(* IEC 61131-3 sources: verifaps-lib/share/PPU.stold (part 8) *)

(* ---- Scenario13_Final.xml_Pusher.st ---- *)
FUNCTION_BLOCK Pusher
    VAR  Duration2 : TIME := TIME#2.0s; END_VAR {*Lrwxp*}
    VAR  Duration3 : TIME := TIME#200.0ms; END_VAR {*Lrwxp*}
    VAR  Duration_Slide1_Black : TIME := TIME#950.0ms; END_VAR {*Lrwxp*}
    VAR  Duration_Slide1_Metal : TIME := TIME#300.0ms; END_VAR {*Lrwxp*}
    VAR  Duration_Slide1_White : TIME := TIME#300.0ms; END_VAR {*Lrwxp*}
    VAR  Duration_Slide2_Black : TIME := TIME#2.0s; END_VAR {*Lrwxp*}
    VAR  Duration_Slide2_Metal : TIME := TIME#370.0ms; END_VAR {*Lrwxp*}
    VAR  Duration_Slide2_White : TIME := TIME#370.0ms; END_VAR {*Lrwxp*}
    VAR  Priority_Var_Black : INT := INT#3; END_VAR {*Lrwxp*}
    VAR  Priority_Var_Metal : INT := INT#3; END_VAR {*Lrwxp*}
    VAR  Priority_Var_White : INT := INT#3; END_VAR {*Lrwxp*}
    VAR_OUTPUT  PusherY1 : BOOL; END_VAR {*Orwxp*}
    VAR_OUTPUT  PusherY2 : BOOL; END_VAR {*Orwxp*}
    VAR  SFCInit : BOOL; END_VAR {*Lrwxp*}
    VAR_INPUT  SFCReset : BOOL; END_VAR {*Irwxp*}
    VAR  Slide1_black : INT := INT#1; END_VAR {*Lrwxp*}
    VAR  Slide1_metal : INT := INT#1; END_VAR {*Lrwxp*}
    VAR  Slide1_white : INT := INT#1; END_VAR {*Lrwxp*}
    VAR  Slide2_black : INT := INT#1; END_VAR {*Lrwxp*}
    VAR  Slide2_metal : INT := INT#1; END_VAR {*Lrwxp*}
    VAR  Slide2_white : INT := INT#1; END_VAR {*Lrwxp*}
    VAR  Slide3_black : INT := INT#1; END_VAR {*Lrwxp*}
    VAR  Slide3_metal : INT := INT#1; END_VAR {*Lrwxp*}
    VAR  Slide3_white : INT := INT#1; END_VAR {*Lrwxp*}
    VAR_INPUT  SorterCapacitiveSensorPusher1 : BOOL; END_VAR {*Irwxp*}
    VAR_INPUT  SorterCapacitiveSensorPusher2 : BOOL; END_VAR {*Irwxp*}
    VAR_INPUT  SorterLightbarrierCraneInterface : BOOL; END_VAR {*Irwxp*}
    VAR_INPUT  SorterLightnessSensorPusher1 : BOOL; END_VAR {*Irwxp*}
    VAR_INPUT  SorterLightnessSensorPusher2 : BOOL; END_VAR {*Irwxp*}
    VAR_INPUT  SorterLightnessSensorPusher3 : BOOL; END_VAR {*Irwxp*}
    VAR_INPUT  SorterLightnesssensorCraneInterfaceInverse : BOOL; END_VAR {*Irwxp*}
    VAR_INPUT  SorterPusher1MovedIn : BOOL; END_VAR {*Irwxp*}
    VAR_INPUT  SorterPusher1MovedOut : BOOL; END_VAR {*Irwxp*}
    VAR_INPUT  SorterPusher2MovedIn : BOOL; END_VAR {*Irwxp*}
    VAR_INPUT  SorterPusher2MovedOut : BOOL; END_VAR {*Irwxp*}
    VAR_INPUT  SorterStartButton : BOOL; END_VAR {*Irwxp*}
    VAR_INPUT  StartVar : BOOL; END_VAR {*Irwxp*}
    VAR  Timer2 : TON; END_VAR {*Lrwxp*}
    VAR  Timer3 : TON; END_VAR {*Lrwxp*}
    VAR  Timer_Slide1_Black : TON; END_VAR {*Lrwxp*}
    VAR  Timer_Slide1_Metal : TON; END_VAR {*Lrwxp*}
    VAR  Timer_Slide1_White : TON; END_VAR {*Lrwxp*}
    VAR  Timer_Slide2_Black : TON; END_VAR {*Lrwxp*}
    VAR  Timer_Slide2_Metal : TON; END_VAR {*Lrwxp*}
    VAR  Timer_Slide2_White : TON; END_VAR {*Lrwxp*}
    VAR  _state : Pusher_states_t; END_VAR {*Lrwxp*}
    VAR  _transit : BOOL; END_VAR {*Lrwxp*}
    VAR  interconnect2 : BOOL; END_VAR {*Lrwxp*}
    VAR  interconnect3 : BOOL; END_VAR {*Lrwxp*}
    VAR  interconnect_Slide1_Black : BOOL; END_VAR {*Lrwxp*}
    VAR  interconnect_Slide1_Metal : BOOL; END_VAR {*Lrwxp*}
    VAR  interconnect_Slide1_White : BOOL; END_VAR {*Lrwxp*}
    VAR  interconnect_Slide2_Black : BOOL; END_VAR {*Lrwxp*}
    VAR  interconnect_Slide2_Metal : BOOL; END_VAR {*Lrwxp*}
    VAR  interconnect_Slide2_White : BOOL; END_VAR {*Lrwxp*}

    CASE _state OF
        Pusher_states_t#Check_For_Black:
            {* begin(State) *}
            {* begin(onEntry) *}
            _transit := FALSE;
            {* end(onEntry) *}
            {* begin(onActive) *}
            {* end(onActive) *}
            {* begin(transition) *}
            IF ((Slide2_black = INT#1) AND (Priority_Var_Black = INT#2)) THEN
                _transit := TRUE;
                _state := Pusher_states_t#Second_Slide_black_workpieces;
            ELSEIF ((Slide3_black = INT#1) AND (Priority_Var_Black = INT#3)) THEN
                _transit := TRUE;
                _state := Pusher_states_t#Third_Slide_black_workpieces;
            ELSEIF ((Slide1_black = INT#1) AND (Priority_Var_Black = INT#1)) THEN
                _transit := TRUE;
                _state := Pusher_states_t#First_Slide_black_workpieces;
            END_IF;
            {* end(transition) *}
            {* begin(onExit) *}
            {* end(onExit) *}
            {* end(State) *}

        Pusher_states_t#Check_For_Metal:
            {* begin(State) *}
            {* begin(onEntry) *}
            _transit := FALSE;
            {* end(onEntry) *}
            {* begin(onActive) *}
            {* end(onActive) *}
            {* begin(transition) *}
            IF ((Slide3_metal = INT#1) AND (Priority_Var_Metal = INT#3)) THEN
                _transit := TRUE;
                _state := Pusher_states_t#Third_Slide_metal_workpieces;
            ELSEIF ((Slide2_metal = INT#1) AND (Priority_Var_Metal = INT#2)) THEN
                _transit := TRUE;
                _state := Pusher_states_t#Second_Slide_metal_workpieces;
            ELSEIF ((Slide1_metal = INT#1) AND (Priority_Var_Metal = INT#1)) THEN
                _transit := TRUE;
                _state := Pusher_states_t#First_Slide_metal_workpieces;
            END_IF;
            {* end(transition) *}
            {* begin(onExit) *}
            {* end(onExit) *}
            {* end(State) *}

        Pusher_states_t#Check_For_White:
            {* begin(State) *}
            {* begin(onEntry) *}
            _transit := FALSE;
            {* end(onEntry) *}
            {* begin(onActive) *}
            {* end(onActive) *}
            {* begin(transition) *}
            IF ((Slide1_white = INT#1) AND (Priority_Var_White = INT#1)) THEN
                _transit := TRUE;
                _state := Pusher_states_t#First_Slide_white_workpieces;
            ELSEIF ((Slide3_white = INT#1) AND (Priority_Var_White = INT#3)) THEN
                _transit := TRUE;
                _state := Pusher_states_t#Third_Slide_white_workpieces;
            ELSEIF ((Slide2_white = INT#1) AND (Priority_Var_White = INT#2)) THEN
                _transit := TRUE;
                _state := Pusher_states_t#Second_Slide_white_workpieces;
            END_IF;
            {* end(transition) *}
            {* begin(onExit) *}
            {* end(onExit) *}
            {* end(State) *}

        Pusher_states_t#First_Slide_Timer_Black:
            {* begin(State) *}
            {* begin(onEntry) *}
            _transit := FALSE;
            {* end(onEntry) *}
            {* begin(onActive) *}
            IF (SorterLightnesssensorCraneInterfaceInverse = TRUE) THEN
                Timer_Slide1_Black(IN := SorterLightnesssensorCraneInterfaceInverse, PT := Duration_Slide1_Black);
                interconnect_Slide1_Black := Timer_Slide1_Black.Q;
            END_IF;
            {* end(onActive) *}
            {* begin(transition) *}
            IF interconnect_Slide1_Black THEN
                _transit := TRUE;
                _state := Pusher_states_t#PusherY1_Move_Out_Black;
            END_IF;
            {* end(transition) *}
            {* begin(onExit) *}
            {* end(onExit) *}
            {* end(State) *}

        Pusher_states_t#First_Slide_Timer_Metal:
            {* begin(State) *}
            {* begin(onEntry) *}
            _transit := FALSE;
            {* end(onEntry) *}
            {* begin(onActive) *}
            Timer_Slide1_Metal(IN := TRUE, PT := Duration_Slide1_Metal);
            interconnect_Slide1_Metal := Timer_Slide1_Metal.Q;
            {* end(onActive) *}
            {* begin(transition) *}
            IF interconnect_Slide1_Metal THEN
                _transit := TRUE;
                _state := Pusher_states_t#PusherY1_Move_Out_Metal;
            END_IF;
            {* end(transition) *}
            {* begin(onExit) *}
            {* end(onExit) *}
            {* end(State) *}

        Pusher_states_t#First_Slide_Timer_White:
            {* begin(State) *}
            {* begin(onEntry) *}
            _transit := FALSE;
            {* end(onEntry) *}
            {* begin(onActive) *}
            Timer_Slide1_White(IN := TRUE, PT := Duration_Slide1_White);
            interconnect_Slide1_White := Timer_Slide1_White.Q;
            {* end(onActive) *}
            {* begin(transition) *}
            IF interconnect_Slide1_White THEN
                _transit := TRUE;
                _state := Pusher_states_t#PusherY1_Move_Out_White;
            END_IF;
            {* end(transition) *}
            {* begin(onExit) *}
            {* end(onExit) *}
            {* end(State) *}

        Pusher_states_t#First_Slide_black_workpieces:
            {* begin(State) *}
            {* begin(onEntry) *}
            _transit := FALSE;
            {* end(onEntry) *}
            {* begin(onActive) *}
            {* end(onActive) *}
            {* begin(transition) *}
            IF TRUE THEN
                _transit := TRUE;
                _state := Pusher_states_t#First_Slide_Timer_Black;
            END_IF;
            {* end(transition) *}
            {* begin(onExit) *}
            {* end(onExit) *}
            {* end(State) *}

        Pusher_states_t#First_Slide_metal_workpieces:
            {* begin(State) *}
            {* begin(onEntry) *}
            _transit := FALSE;
            {* end(onEntry) *}
            {* begin(onActive) *}
            {* end(onActive) *}
            {* begin(transition) *}
            IF TRUE THEN
                _transit := TRUE;
                _state := Pusher_states_t#First_Slide_Timer_Metal;
            END_IF;
            {* end(transition) *}
            {* begin(onExit) *}
            {* end(onExit) *}
            {* end(State) *}

        Pusher_states_t#First_Slide_white_workpieces:
            {* begin(State) *}
            {* begin(onEntry) *}
            _transit := FALSE;
            {* end(onEntry) *}
            {* begin(onActive) *}
            {* end(onActive) *}
            {* begin(transition) *}
            IF TRUE THEN
                _transit := TRUE;
                _state := Pusher_states_t#First_Slide_Timer_White;
            END_IF;
            {* end(transition) *}
            {* begin(onExit) *}
            {* end(onExit) *}
            {* end(State) *}

        Pusher_states_t#Init:
            {* begin(State) *}
            {* begin(onEntry) *}
            _transit := FALSE;
            {* end(onEntry) *}
            {* begin(onActive) *}
            {* end(onActive) *}
            {* begin(transition) *}
            IF StartVar THEN
                _transit := TRUE;
                _state := Pusher_states_t#Interstep;
            END_IF;
            {* end(transition) *}
            {* begin(onExit) *}
            {* end(onExit) *}
            {* end(State) *}

        Pusher_states_t#Interstep:
            {* begin(State) *}
            {* begin(onEntry) *}
            _transit := FALSE;
            {* end(onEntry) *}
            {* begin(onActive) *}
            PusherY1 := FALSE;
            PusherY2 := FALSE;
            interconnect2 := FALSE;
            interconnect3 := FALSE;
            StartVar := FALSE;
            interconnect_Slide1_Black := FALSE;
            interconnect_Slide2_Black := FALSE;
            interconnect_Slide1_White := FALSE;
            interconnect_Slide2_White := FALSE;
            interconnect_Slide1_Metal := FALSE;
            interconnect_Slide2_Metal := FALSE;
            {* end(onActive) *}
            {* begin(transition) *}
            IF TRUE THEN
                _transit := TRUE;
                _state := Pusher_states_t#Interstep_2;
            END_IF;
            {* end(transition) *}
            {* begin(onExit) *}
            {* end(onExit) *}
            {* end(State) *}

        Pusher_states_t#Interstep_2:
            {* begin(State) *}
            {* begin(onEntry) *}
            _transit := FALSE;
            {* end(onEntry) *}
            {* begin(onActive) *}
            {* end(onActive) *}
            {* begin(transition) *}
            IF ((SorterLightnessSensorPusher1 AND SorterCapacitiveSensorPusher1) AND (Priority_Var_Metal > INT#0)) THEN
                _transit := TRUE;
                _state := Pusher_states_t#Check_For_Metal;
            ELSEIF ((NOT SorterLightnesssensorCraneInterfaceInverse AND SorterLightbarrierCraneInterface) AND (Priority_Var_Black > INT#0)) THEN
                _transit := TRUE;
                _state := Pusher_states_t#Check_For_Black;
            ELSEIF ((SorterLightnessSensorPusher1 AND NOT SorterCapacitiveSensorPusher1) AND (Priority_Var_White > INT#0)) THEN
                _transit := TRUE;
                _state := Pusher_states_t#Check_For_White;
            END_IF;
            {* end(transition) *}
            {* begin(onExit) *}
            {* end(onExit) *}
            {* end(State) *}

        Pusher_states_t#PusherY1_Move_In_Black:
            {* begin(State) *}
            {* begin(onEntry) *}
            _transit := FALSE;
            {* end(onEntry) *}
            {* begin(onActive) *}
            IF ((SorterPusher1MovedOut = TRUE) AND (SorterPusher1MovedIn = FALSE)) THEN
                PusherY1 := FALSE;
            END_IF;
            {* end(onActive) *}
            {* begin(transition) *}
            IF SorterPusher1MovedIn THEN
                _transit := TRUE;
                _state := Pusher_states_t#Reset_interconnect_Slide1_Black;
            END_IF;
            {* end(transition) *}
            {* begin(onExit) *}
            {* end(onExit) *}
            {* end(State) *}

        Pusher_states_t#PusherY1_Move_In_Metal:
            {* begin(State) *}
            {* begin(onEntry) *}
            _transit := FALSE;
            {* end(onEntry) *}
            {* begin(onActive) *}
            IF ((SorterPusher1MovedOut = TRUE) AND (SorterPusher1MovedIn = FALSE)) THEN
                PusherY1 := FALSE;
            END_IF;
            {* end(onActive) *}
            {* begin(transition) *}
            IF SorterPusher1MovedIn THEN
                _transit := TRUE;
                _state := Pusher_states_t#Reset_interconnect_Slide1_Metal;
            END_IF;
            {* end(transition) *}
            {* begin(onExit) *}
            {* end(onExit) *}
            {* end(State) *}

        Pusher_states_t#PusherY1_Move_In_White:
            {* begin(State) *}
            {* begin(onEntry) *}
            _transit := FALSE;
            {* end(onEntry) *}
            {* begin(onActive) *}
            IF ((SorterPusher1MovedOut = TRUE) AND (SorterPusher1MovedIn = FALSE)) THEN
                PusherY1 := FALSE;
            END_IF;
            {* end(onActive) *}
            {* begin(transition) *}
            IF SorterPusher1MovedIn THEN
                _transit := TRUE;
                _state := Pusher_states_t#Reset_interconnect_Slide1_White;
            END_IF;
            {* end(transition) *}
            {* begin(onExit) *}
            {* end(onExit) *}
            {* end(State) *}

        Pusher_states_t#PusherY1_Move_Out_Black:
            {* begin(State) *}
            {* begin(onEntry) *}
            _transit := FALSE;
            {* end(onEntry) *}
            {* begin(onActive) *}
            IF ((SorterPusher1MovedOut = FALSE) AND (SorterPusher1MovedIn = TRUE)) THEN
                PusherY1 := TRUE;
            END_IF;
            {* end(onActive) *}
            {* begin(transition) *}
            IF SorterPusher1MovedOut THEN
                _transit := TRUE;
                _state := Pusher_states_t#Wait_Y1_Black;
            END_IF;
            {* end(transition) *}
            {* begin(onExit) *}
            {* end(onExit) *}
            {* end(State) *}

        Pusher_states_t#PusherY1_Move_Out_Metal:
            {* begin(State) *}
            {* begin(onEntry) *}
            _transit := FALSE;
            {* end(onEntry) *}
            {* begin(onActive) *}
            IF ((SorterPusher1MovedOut = FALSE) AND (SorterPusher1MovedIn = TRUE)) THEN
                PusherY1 := TRUE;
            END_IF;
            {* end(onActive) *}
            {* begin(transition) *}
            IF SorterPusher1MovedOut THEN
                _transit := TRUE;
                _state := Pusher_states_t#Wait_Y1_Metal;
            END_IF;
            {* end(transition) *}
            {* begin(onExit) *}
            {* end(onExit) *}
            {* end(State) *}

        Pusher_states_t#PusherY1_Move_Out_White:
            {* begin(State) *}
            {* begin(onEntry) *}
            _transit := FALSE;
            {* end(onEntry) *}
            {* begin(onActive) *}
            IF ((SorterPusher1MovedOut = FALSE) AND (SorterPusher1MovedIn = TRUE)) THEN
                PusherY1 := TRUE;
            END_IF;
            {* end(onActive) *}
            {* begin(transition) *}
            IF SorterPusher1MovedOut THEN
                _transit := TRUE;
                _state := Pusher_states_t#Wait_Y1_White;
            END_IF;
            {* end(transition) *}
            {* begin(onExit) *}
            {* end(onExit) *}
            {* end(State) *}

        Pusher_states_t#PusherY2_Move_In_Black:
            {* begin(State) *}
            {* begin(onEntry) *}
            _transit := FALSE;
            {* end(onEntry) *}
            {* begin(onActive) *}
            IF ((SorterPusher2MovedOut = TRUE) AND (SorterPusher2MovedIn = FALSE)) THEN
                PusherY2 := FALSE;
            END_IF;
            {* end(onActive) *}
            {* begin(transition) *}
            IF SorterPusher2MovedIn THEN
                _transit := TRUE;
                _state := Pusher_states_t#Reset_interconnect_Slide2_Black;
            END_IF;
            {* end(transition) *}
            {* begin(onExit) *}
            {* end(onExit) *}
            {* end(State) *}

        Pusher_states_t#PusherY2_Move_In_Metal:
            {* begin(State) *}
            {* begin(onEntry) *}
            _transit := FALSE;
            {* end(onEntry) *}
            {* begin(onActive) *}
            IF ((SorterPusher2MovedOut = TRUE) AND (SorterPusher2MovedIn = FALSE)) THEN
                PusherY2 := FALSE;
            END_IF;
            {* end(onActive) *}
            {* begin(transition) *}
            IF SorterPusher2MovedIn THEN
                _transit := TRUE;
                _state := Pusher_states_t#Reset_interconnect_Slide2_Metal;
            END_IF;
            {* end(transition) *}
            {* begin(onExit) *}
            {* end(onExit) *}
            {* end(State) *}

        Pusher_states_t#PusherY2_Move_In_White:
            {* begin(State) *}
            {* begin(onEntry) *}
            _transit := FALSE;
            {* end(onEntry) *}
            {* begin(onActive) *}
            IF ((SorterPusher2MovedOut = TRUE) AND (SorterPusher2MovedIn = FALSE)) THEN
                PusherY2 := FALSE;
            END_IF;
            {* end(onActive) *}
            {* begin(transition) *}
            IF SorterPusher2MovedIn THEN
                _transit := TRUE;
                _state := Pusher_states_t#Reset_interconnect_Slide2_White;
            END_IF;
            {* end(transition) *}
            {* begin(onExit) *}
            {* end(onExit) *}
            {* end(State) *}

        Pusher_states_t#PusherY2_Move_Out_Black:
            {* begin(State) *}
            {* begin(onEntry) *}
            _transit := FALSE;
            {* end(onEntry) *}
            {* begin(onActive) *}
            IF ((SorterPusher2MovedOut = FALSE) AND (SorterPusher2MovedIn = TRUE)) THEN
                PusherY2 := TRUE;
            END_IF;
            {* end(onActive) *}
            {* begin(transition) *}
            IF SorterPusher2MovedOut THEN
                _transit := TRUE;
                _state := Pusher_states_t#Wait_Y2_Black;
            END_IF;
            {* end(transition) *}
            {* begin(onExit) *}
            {* end(onExit) *}
            {* end(State) *}

        Pusher_states_t#PusherY2_Move_Out_Metal:
            {* begin(State) *}
            {* begin(onEntry) *}
            _transit := FALSE;
            {* end(onEntry) *}
            {* begin(onActive) *}
            IF ((SorterPusher2MovedOut = FALSE) AND (SorterPusher2MovedIn = TRUE)) THEN
                PusherY2 := TRUE;
            END_IF;
            {* end(onActive) *}
            {* begin(transition) *}
            IF SorterPusher2MovedOut THEN
                _transit := TRUE;
                _state := Pusher_states_t#Wait_Y2_Metal;
            END_IF;
            {* end(transition) *}
            {* begin(onExit) *}
            {* end(onExit) *}
            {* end(State) *}

        Pusher_states_t#PusherY2_Move_Out_White:
            {* begin(State) *}
            {* begin(onEntry) *}
            _transit := FALSE;
            {* end(onEntry) *}
            {* begin(onActive) *}
            IF ((SorterPusher2MovedOut = FALSE) AND (SorterPusher2MovedIn = TRUE)) THEN
                PusherY2 := TRUE;
            END_IF;
            {* end(onActive) *}
            {* begin(transition) *}
            IF SorterPusher2MovedOut THEN
                _transit := TRUE;
                _state := Pusher_states_t#Wait_Y2_White;
            END_IF;
            {* end(transition) *}
            {* begin(onExit) *}
            {* end(onExit) *}
            {* end(State) *}

        Pusher_states_t#Reset_interconnect3:
            {* begin(State) *}
            {* begin(onEntry) *}
            _transit := FALSE;
            {* end(onEntry) *}
            {* begin(onActive) *}
            interconnect2 := FALSE;
            Timer2(IN := FALSE, PT := TIME#);
            Slide3_black := (Slide3_black - INT#1);
            Priority_Var_Black := (Priority_Var_Black - INT#1);
            {* end(onActive) *}
            {* begin(transition) *}
            IF TRUE THEN
                _transit := TRUE;
                _state := Pusher_states_t#Interstep_2;
            END_IF;
            {* end(transition) *}
            {* begin(onExit) *}
            {* end(onExit) *}
            {* end(State) *}

        Pusher_states_t#Reset_interconnect_Slide1_Black:
            {* begin(State) *}
            {* begin(onEntry) *}
            _transit := FALSE;
            {* end(onEntry) *}
            {* begin(onActive) *}
            interconnect3 := FALSE;
            Timer3(IN := FALSE, PT := TIME#);
            interconnect_Slide1_Black := FALSE;
            Timer_Slide1_Black(IN := FALSE, PT := TIME#);
            Slide1_black := (Slide1_black - INT#1);
            Priority_Var_Black := (Priority_Var_Black - INT#1);
            {* end(onActive) *}
            {* begin(transition) *}
            IF TRUE THEN
                _transit := TRUE;
                _state := Pusher_states_t#Interstep_2;
            END_IF;
            {* end(transition) *}
            {* begin(onExit) *}
            {* end(onExit) *}
            {* end(State) *}

        Pusher_states_t#Reset_interconnect_Slide1_Metal:
            {* begin(State) *}
            {* begin(onEntry) *}
            _transit := FALSE;
            {* end(onEntry) *}
            {* begin(onActive) *}
            interconnect3 := FALSE;
            Timer3(IN := FALSE, PT := TIME#);
            interconnect_Slide1_Metal := FALSE;
            Timer_Slide1_Metal(IN := FALSE, PT := TIME#);
            Slide1_metal := (Slide1_metal - INT#1);
            Priority_Var_Metal := (Priority_Var_Metal - INT#1);
            {* end(onActive) *}
            {* begin(transition) *}
            IF TRUE THEN
                _transit := TRUE;
                _state := Pusher_states_t#Interstep_2;
            END_IF;
            {* end(transition) *}
            {* begin(onExit) *}
            {* end(onExit) *}
            {* end(State) *}

        Pusher_states_t#Reset_interconnect_Slide1_White:
            {* begin(State) *}
            {* begin(onEntry) *}
            _transit := FALSE;
            {* end(onEntry) *}
            {* begin(onActive) *}
            interconnect3 := FALSE;
            Timer3(IN := FALSE, PT := TIME#);
            interconnect_Slide1_White := FALSE;
            Timer_Slide1_White(IN := FALSE, PT := TIME#);
            Slide1_white := (Slide1_white - INT#1);
            Priority_Var_White := (Priority_Var_White - INT#1);
            {* end(onActive) *}
            {* begin(transition) *}
            IF TRUE THEN
                _transit := TRUE;
                _state := Pusher_states_t#Interstep_2;
            END_IF;
            {* end(transition) *}
            {* begin(onExit) *}
            {* end(onExit) *}
            {* end(State) *}

        Pusher_states_t#Reset_interconnect_Slide2_Black:
            {* begin(State) *}
            {* begin(onEntry) *}
            _transit := FALSE;
            {* end(onEntry) *}
            {* begin(onActive) *}
            interconnect3 := FALSE;
            Timer3(IN := FALSE, PT := TIME#);
            interconnect_Slide2_Black := FALSE;
            Timer_Slide2_Black(IN := FALSE, PT := TIME#);
            Slide2_black := (Slide2_black - INT#1);
            Priority_Var_Black := (Priority_Var_Black - INT#1);
            {* end(onActive) *}
            {* begin(transition) *}
            IF TRUE THEN
                _transit := TRUE;
                _state := Pusher_states_t#Interstep_2;
            END_IF;
            {* end(transition) *}
            {* begin(onExit) *}
            {* end(onExit) *}
            {* end(State) *}

        Pusher_states_t#Reset_interconnect_Slide2_Metal:
            {* begin(State) *}
            {* begin(onEntry) *}
            _transit := FALSE;
            {* end(onEntry) *}
            {* begin(onActive) *}
            interconnect3 := FALSE;
            Timer3(IN := FALSE, PT := TIME#);
            interconnect_Slide2_Metal := FALSE;
            Timer_Slide2_Metal(IN := FALSE, PT := TIME#);
            Slide2_metal := (Slide2_metal - INT#1);
            Priority_Var_Metal := (Priority_Var_Metal - INT#1);
            {* end(onActive) *}
            {* begin(transition) *}
            IF TRUE THEN
                _transit := TRUE;
                _state := Pusher_states_t#Interstep_2;
            END_IF;
            {* end(transition) *}
            {* begin(onExit) *}
            {* end(onExit) *}
            {* end(State) *}

        Pusher_states_t#Reset_interconnect_Slide2_White:
            {* begin(State) *}
            {* begin(onEntry) *}
            _transit := FALSE;
            {* end(onEntry) *}
            {* begin(onActive) *}
            interconnect3 := FALSE;
            Timer3(IN := FALSE, PT := TIME#);
            interconnect_Slide2_White := FALSE;
            Timer_Slide2_White(IN := FALSE, PT := TIME#);
            Slide2_white := (Slide2_white - INT#1);
            Priority_Var_White := (Priority_Var_White - INT#1);
            {* end(onActive) *}
            {* begin(transition) *}
            IF TRUE THEN
                _transit := TRUE;
                _state := Pusher_states_t#Interstep_2;
            END_IF;
            {* end(transition) *}
            {* begin(onExit) *}
            {* end(onExit) *}
            {* end(State) *}

        Pusher_states_t#Reset_interconnect_Slide3_Metal:
            {* begin(State) *}
            {* begin(onEntry) *}
            _transit := FALSE;
            {* end(onEntry) *}
            {* begin(onActive) *}
            interconnect3 := FALSE;
            Timer3(IN := FALSE, PT := TIME#);
            Slide3_metal := (Slide3_metal - INT#1);
            Priority_Var_Metal := (Priority_Var_Metal - INT#1);
            {* end(onActive) *}
            {* begin(transition) *}
            IF TRUE THEN
                _transit := TRUE;
                _state := Pusher_states_t#Interstep_2;
            END_IF;
            {* end(transition) *}
            {* begin(onExit) *}
            {* end(onExit) *}
            {* end(State) *}

        Pusher_states_t#Reset_interconnect_Slide3_White:
            {* begin(State) *}
            {* begin(onEntry) *}
            _transit := FALSE;
            {* end(onEntry) *}
            {* begin(onActive) *}
            interconnect3 := FALSE;
            Timer3(IN := FALSE, PT := TIME#);
            Slide3_white := (Slide3_white - INT#1);
            Priority_Var_White := (Priority_Var_White - INT#1);
            {* end(onActive) *}
            {* begin(transition) *}
            IF TRUE THEN
                _transit := TRUE;
                _state := Pusher_states_t#Interstep_2;
            END_IF;
            {* end(transition) *}
            {* begin(onExit) *}
            {* end(onExit) *}
            {* end(State) *}

        Pusher_states_t#Second_Slide_Timer_Black:
            {* begin(State) *}
            {* begin(onEntry) *}
            _transit := FALSE;
            {* end(onEntry) *}
            {* begin(onActive) *}
            IF (SorterLightnesssensorCraneInterfaceInverse = TRUE) THEN
                Timer_Slide2_Black(IN := SorterLightnesssensorCraneInterfaceInverse, PT := Duration_Slide2_Black);
                interconnect_Slide2_Black := Timer_Slide2_Black.Q;
            END_IF;
            {* end(onActive) *}
            {* begin(transition) *}
            IF interconnect_Slide2_Black THEN
                _transit := TRUE;
                _state := Pusher_states_t#PusherY2_Move_Out_Black;
            END_IF;
            {* end(transition) *}
            {* begin(onExit) *}
            {* end(onExit) *}
            {* end(State) *}

        Pusher_states_t#Second_Slide_Timer_Metal:
            {* begin(State) *}
            {* begin(onEntry) *}
            _transit := FALSE;
            {* end(onEntry) *}
            {* begin(onActive) *}
            Timer_Slide2_Metal(IN := TRUE, PT := Duration_Slide2_Metal);
            interconnect_Slide2_Metal := Timer_Slide2_Metal.Q;
            {* end(onActive) *}
            {* begin(transition) *}
            IF interconnect_Slide2_Metal THEN
                _transit := TRUE;
                _state := Pusher_states_t#PusherY2_Move_Out_Metal;
            END_IF;
            {* end(transition) *}
            {* begin(onExit) *}
            {* end(onExit) *}
            {* end(State) *}

        Pusher_states_t#Second_Slide_Timer_White:
            {* begin(State) *}
            {* begin(onEntry) *}
            _transit := FALSE;
            {* end(onEntry) *}
            {* begin(onActive) *}
            Timer_Slide2_White(IN := TRUE, PT := Duration_Slide2_White);
            interconnect_Slide2_White := Timer_Slide2_White.Q;
            {* end(onActive) *}
            {* begin(transition) *}
            IF interconnect_Slide2_White THEN
                _transit := TRUE;
                _state := Pusher_states_t#PusherY2_Move_Out_White;
            END_IF;
            {* end(transition) *}
            {* begin(onExit) *}
            {* end(onExit) *}
            {* end(State) *}

        Pusher_states_t#Second_Slide_black_workpieces:
            {* begin(State) *}
            {* begin(onEntry) *}
            _transit := FALSE;
            {* end(onEntry) *}
            {* begin(onActive) *}
            {* end(onActive) *}
            {* begin(transition) *}
            IF TRUE THEN
                _transit := TRUE;
                _state := Pusher_states_t#Second_Slide_Timer_Black;
            END_IF;
            {* end(transition) *}
            {* begin(onExit) *}
            {* end(onExit) *}
            {* end(State) *}

        Pusher_states_t#Second_Slide_metal_workpieces:
            {* begin(State) *}
            {* begin(onEntry) *}
            _transit := FALSE;
            {* end(onEntry) *}
            {* begin(onActive) *}
            {* end(onActive) *}
            {* begin(transition) *}
            IF (SorterLightnessSensorPusher2 AND SorterCapacitiveSensorPusher2) THEN
                _transit := TRUE;
                _state := Pusher_states_t#Second_Test_For_Metal;
            END_IF;
            {* end(transition) *}
            {* begin(onExit) *}
            {* end(onExit) *}
            {* end(State) *}

        Pusher_states_t#Second_Slide_white_workpieces:
            {* begin(State) *}
            {* begin(onEntry) *}
            _transit := FALSE;
            {* end(onEntry) *}
            {* begin(onActive) *}
            {* end(onActive) *}
            {* begin(transition) *}
            IF (SorterLightnessSensorPusher2 AND NOT SorterCapacitiveSensorPusher2) THEN
                _transit := TRUE;
                _state := Pusher_states_t#Second_Test_For_White;
            END_IF;
            {* end(transition) *}
            {* begin(onExit) *}
            {* end(onExit) *}
            {* end(State) *}

        Pusher_states_t#Second_Test_For_Metal:
            {* begin(State) *}
            {* begin(onEntry) *}
            _transit := FALSE;
            {* end(onEntry) *}
            {* begin(onActive) *}
            {* end(onActive) *}
            {* begin(transition) *}
            IF TRUE THEN
                _transit := TRUE;
                _state := Pusher_states_t#Second_Slide_Timer_Metal;
            END_IF;
            {* end(transition) *}
            {* begin(onExit) *}
            {* end(onExit) *}
            {* end(State) *}

        Pusher_states_t#Second_Test_For_White:
            {* begin(State) *}
            {* begin(onEntry) *}
            _transit := FALSE;
            {* end(onEntry) *}
            {* begin(onActive) *}
            {* end(onActive) *}
            {* begin(transition) *}
            IF TRUE THEN
                _transit := TRUE;
                _state := Pusher_states_t#Second_Slide_Timer_White;
            END_IF;
            {* end(transition) *}
            {* begin(onExit) *}
            {* end(onExit) *}
            {* end(State) *}

        Pusher_states_t#Third_Slide_black_workpieces:
            {* begin(State) *}
            {* begin(onEntry) *}
            _transit := FALSE;
            {* end(onEntry) *}
            {* begin(onActive) *}
            {* end(onActive) *}
            {* begin(transition) *}
            IF (NOT SorterLightnessSensorPusher2 AND NOT SorterCapacitiveSensorPusher2) THEN
                _transit := TRUE;
                _state := Pusher_states_t#Wait_Black;
            END_IF;
            {* end(transition) *}
            {* begin(onExit) *}
            {* end(onExit) *}
            {* end(State) *}

        Pusher_states_t#Third_Slide_metal_workpieces:
            {* begin(State) *}
            {* begin(onEntry) *}
            _transit := FALSE;
            {* end(onEntry) *}
            {* begin(onActive) *}
            {* end(onActive) *}
            {* begin(transition) *}
            IF (SorterLightnessSensorPusher2 AND SorterCapacitiveSensorPusher2) THEN
                _transit := TRUE;
                _state := Pusher_states_t#Wait_Metal;
            END_IF;
            {* end(transition) *}
            {* begin(onExit) *}
            {* end(onExit) *}
            {* end(State) *}

        Pusher_states_t#Third_Slide_white_workpieces:
            {* begin(State) *}
            {* begin(onEntry) *}
            _transit := FALSE;
            {* end(onEntry) *}
            {* begin(onActive) *}
            {* end(onActive) *}
            {* begin(transition) *}
            IF (SorterLightnessSensorPusher2 AND NOT SorterCapacitiveSensorPusher2) THEN
                _transit := TRUE;
                _state := Pusher_states_t#Wait_White;
            END_IF;
            {* end(transition) *}
            {* begin(onExit) *}
            {* end(onExit) *}
            {* end(State) *}

        Pusher_states_t#Wait_Black:
            {* begin(State) *}
            {* begin(onEntry) *}
            _transit := FALSE;
            {* end(onEntry) *}
            {* begin(onActive) *}
            IF ((NOT SorterLightnessSensorPusher2 AND NOT SorterCapacitiveSensorPusher2) = TRUE) THEN
                Timer2(IN := (NOT SorterLightnessSensorPusher2 AND NOT SorterCapacitiveSensorPusher2), PT := Duration2);
                interconnect2 := Timer2.Q;
            END_IF;
            {* end(onActive) *}
            {* begin(transition) *}
            IF interconnect2 THEN
                _transit := TRUE;
                _state := Pusher_states_t#Reset_interconnect3;
            END_IF;
            {* end(transition) *}
            {* begin(onExit) *}
            {* end(onExit) *}
            {* end(State) *}

        Pusher_states_t#Wait_Metal:
            {* begin(State) *}
            {* begin(onEntry) *}
            _transit := FALSE;
            {* end(onEntry) *}
            {* begin(onActive) *}
            Timer3(IN := TRUE, PT := Duration3);
            interconnect3 := Timer3.Q;
            {* end(onActive) *}
            {* begin(transition) *}
            IF interconnect3 THEN
                _transit := TRUE;
                _state := Pusher_states_t#Reset_interconnect_Slide3_Metal;
            END_IF;
            {* end(transition) *}
            {* begin(onExit) *}
            {* end(onExit) *}
            {* end(State) *}

        Pusher_states_t#Wait_White:
            {* begin(State) *}
            {* begin(onEntry) *}
            _transit := FALSE;
            {* end(onEntry) *}
            {* begin(onActive) *}
            Timer3(IN := TRUE, PT := Duration3);
            interconnect3 := Timer3.Q;
            {* end(onActive) *}
            {* begin(transition) *}
            IF interconnect3 THEN
                _transit := TRUE;
                _state := Pusher_states_t#Reset_interconnect_Slide3_White;
            END_IF;
            {* end(transition) *}
            {* begin(onExit) *}
            {* end(onExit) *}
            {* end(State) *}

        Pusher_states_t#Wait_Y1_Black:
            {* begin(State) *}
            {* begin(onEntry) *}
            _transit := FALSE;
            {* end(onEntry) *}
            {* begin(onActive) *}
            IF (PusherY1 = TRUE) THEN
                Timer3(IN := PusherY1, PT := Duration3);
                interconnect3 := Timer3.Q;
            END_IF;
            {* end(onActive) *}
            {* begin(transition) *}
            IF interconnect3 THEN
                _transit := TRUE;
                _state := Pusher_states_t#PusherY1_Move_In_Black;
            END_IF;
            {* end(transition) *}
            {* begin(onExit) *}
            {* end(onExit) *}
            {* end(State) *}

        Pusher_states_t#Wait_Y1_Metal:
            {* begin(State) *}
            {* begin(onEntry) *}
            _transit := FALSE;
            {* end(onEntry) *}
            {* begin(onActive) *}
            IF (PusherY1 = TRUE) THEN
                Timer3(IN := PusherY1, PT := Duration3);
                interconnect3 := Timer3.Q;
            END_IF;
            {* end(onActive) *}
            {* begin(transition) *}
            IF interconnect3 THEN
                _transit := TRUE;
                _state := Pusher_states_t#PusherY1_Move_In_Metal;
            END_IF;
            {* end(transition) *}
            {* begin(onExit) *}
            {* end(onExit) *}
            {* end(State) *}

        Pusher_states_t#Wait_Y1_White:
            {* begin(State) *}
            {* begin(onEntry) *}
            _transit := FALSE;
            {* end(onEntry) *}
            {* begin(onActive) *}
            IF (PusherY1 = TRUE) THEN
                Timer3(IN := PusherY1, PT := Duration3);
                interconnect3 := Timer3.Q;
            END_IF;
            {* end(onActive) *}
            {* begin(transition) *}
            IF interconnect3 THEN
                _transit := TRUE;
                _state := Pusher_states_t#PusherY1_Move_In_White;
            END_IF;
            {* end(transition) *}
            {* begin(onExit) *}
            {* end(onExit) *}
            {* end(State) *}

        Pusher_states_t#Wait_Y2_Black:
            {* begin(State) *}
            {* begin(onEntry) *}
            _transit := FALSE;
            {* end(onEntry) *}
            {* begin(onActive) *}
            IF (PusherY2 = TRUE) THEN
                Timer3(IN := PusherY2, PT := Duration3);
                interconnect3 := Timer3.Q;
            END_IF;
            {* end(onActive) *}
            {* begin(transition) *}
            IF interconnect3 THEN
                _transit := TRUE;
                _state := Pusher_states_t#PusherY2_Move_In_Black;
            END_IF;
            {* end(transition) *}
            {* begin(onExit) *}
            {* end(onExit) *}
            {* end(State) *}

        Pusher_states_t#Wait_Y2_Metal:
            {* begin(State) *}
            {* begin(onEntry) *}
            _transit := FALSE;
            {* end(onEntry) *}
            {* begin(onActive) *}
            IF (PusherY2 = TRUE) THEN
                Timer3(IN := PusherY2, PT := Duration3);
                interconnect3 := Timer3.Q;
            END_IF;
            {* end(onActive) *}
            {* begin(transition) *}
            IF interconnect3 THEN
                _transit := TRUE;
                _state := Pusher_states_t#PusherY2_Move_In_Metal;
            END_IF;
            {* end(transition) *}
            {* begin(onExit) *}
            {* end(onExit) *}
            {* end(State) *}

        Pusher_states_t#Wait_Y2_White:
            {* begin(State) *}
            {* begin(onEntry) *}
            _transit := FALSE;
            {* end(onEntry) *}
            {* begin(onActive) *}
            IF (PusherY2 = TRUE) THEN
                Timer3(IN := PusherY2, PT := Duration3);
                interconnect3 := Timer3.Q;
            END_IF;
            {* end(onActive) *}
            {* begin(transition) *}
            IF interconnect3 THEN
                _transit := TRUE;
                _state := Pusher_states_t#PusherY2_Move_In_White;
            END_IF;
            {* end(transition) *}
            {* begin(onExit) *}
            {* end(onExit) *}
            {* end(State) *}

            END_CASE;
END_FUNCTION_BLOCK

(* ---- Scenario13_Final.xml_Stamp.st ---- *)
FUNCTION_BLOCK Stamp
    VAR_INPUT  AnalogCranePosition : INT; END_VAR {*Irwxp*}
    VAR_INPUT  CraneDown : BOOL; END_VAR {*Irwxp*}
    VAR_INPUT  CraneOnConveyor : BOOL; END_VAR {*Irwxp*}
    VAR_INPUT  CranePositionStamp : BOOL; END_VAR {*Irwxp*}
    VAR_INPUT  CraneSucked : BOOL; END_VAR {*Irwxp*}
    VAR_INPUT  CraneUp : BOOL; END_VAR {*Irwxp*}
    VAR  Duration : TIME := TIME#500.0ms; END_VAR {*Lrwxp*}
    VAR  SFCInit : BOOL; END_VAR {*Lrwxp*}
    VAR_INPUT  SFCReset : BOOL; END_VAR {*Irwxp*}
    VAR_OUTPUT  StampGreenLamp : BOOL; END_VAR {*Orwxp*}
    VAR_INPUT  StampLowered : BOOL; END_VAR {*Irwxp*}
    VAR_OUTPUT  StampPressure : BOOL; END_VAR {*Orwxp*}
    VAR_OUTPUT  StampPusher : BOOL; END_VAR {*Orwxp*}
    VAR_INPUT  StampSliderFilled : BOOL; END_VAR {*Irwxp*}
    VAR_OUTPUT  StampSliderMovedIn : BOOL; END_VAR {*Orwxp*}
    VAR_OUTPUT  StampSliderMovedOut : BOOL; END_VAR {*Orwxp*}
    VAR_INPUT  StampSliderSensorMovedIn : BOOL; END_VAR {*Irwxp*}
    VAR_INPUT  StampSliderSensorMovedOut : BOOL; END_VAR {*Irwxp*}
    VAR_INPUT  StampStartButton : BOOL; END_VAR {*Irwxp*}
    VAR_INPUT  StampUp : BOOL; END_VAR {*Irwxp*}
    VAR_OUTPUT  StampWhiteLamp : BOOL; END_VAR {*Orwxp*}
    VAR_OUTPUT  StartCommandStamp : BOOL; END_VAR {*Orwxp*}
    VAR_INPUT  StartVar : BOOL; END_VAR {*Irwxp*}
    VAR  Timer : TON; END_VAR {*Lrwxp*}
    VAR  _state : Stamp_states_t; END_VAR {*Lrwxp*}
    VAR  _transit : BOOL; END_VAR {*Lrwxp*}
    VAR  interconnect : BOOL; END_VAR {*Lrwxp*}
    VAR  interconnectStampStartCommand : BOOL; END_VAR {*Lrwxp*}

    CASE _state OF
        Stamp_states_t#Green_Lamp:
            {* begin(State) *}
            {* begin(onEntry) *}
            _transit := FALSE;
            {* end(onEntry) *}
            {* begin(onActive) *}
            StampGreenLamp := TRUE;
            interconnectStampStartCommand := FALSE;
            {* end(onActive) *}
            {* begin(transition) *}
            IF TRUE THEN
                _transit := TRUE;
                _state := Stamp_states_t#Stamp_Init_1;
            END_IF;
            {* end(transition) *}
            {* begin(onExit) *}
            {* end(onExit) *}
            {* end(State) *}

        Stamp_states_t#Init:
            {* begin(State) *}
            {* begin(onEntry) *}
            _transit := FALSE;
            {* end(onEntry) *}
            {* begin(onActive) *}
            {* end(onActive) *}
            {* begin(transition) *}
            IF TRUE THEN
                _transit := TRUE;
                _state := Stamp_states_t#Start_Stamp;
            END_IF;
            {* end(transition) *}
            {* begin(onExit) *}
            {* end(onExit) *}
            {* end(State) *}

        Stamp_states_t#Interstep:
            {* begin(State) *}
            {* begin(onEntry) *}
            _transit := FALSE;
            {* end(onEntry) *}
            {* begin(onActive) *}
            StartCommandStamp := TRUE;
            {* end(onActive) *}
            {* begin(transition) *}
            IF StartVar THEN
                _transit := TRUE;
                _state := Stamp_states_t#Intertsep_2;
            END_IF;
            {* end(transition) *}
            {* begin(onExit) *}
            {* end(onExit) *}
            {* end(State) *}

        Stamp_states_t#Intertsep_2:
            {* begin(State) *}
            {* begin(onEntry) *}
            _transit := FALSE;
            {* end(onEntry) *}
            {* begin(onActive) *}
            {* end(onActive) *}
            {* begin(transition) *}
            IF StampSliderFilled THEN
                _transit := TRUE;
                _state := Stamp_states_t#Step0;
            END_IF;
            {* end(transition) *}
            {* begin(onExit) *}
            {* end(onExit) *}
            {* end(State) *}

        Stamp_states_t#StampProcess:
            {* begin(State) *}
            {* begin(onEntry) *}
            _transit := FALSE;
            {* end(onEntry) *}
            {* begin(onActive) *}
            StampSliderMovedIn := FALSE;
            StampPusher := TRUE;
            {* end(onActive) *}
            {* begin(transition) *}
            IF StampLowered THEN
                _transit := TRUE;
                _state := Stamp_states_t#Step1;
            END_IF;
            {* end(transition) *}
            {* begin(onExit) *}
            {* end(onExit) *}
            {* end(State) *}

        Stamp_states_t#StampSliderBack:
            {* begin(State) *}
            {* begin(onEntry) *}
            _transit := FALSE;
            {* end(onEntry) *}
            {* begin(onActive) *}
            StampSliderMovedIn := TRUE;
            StampSliderMovedOut := FALSE;
            {* end(onActive) *}
            {* begin(transition) *}
            IF StampSliderSensorMovedIn THEN
                _transit := TRUE;
                _state := Stamp_states_t#StampProcess;
            END_IF;
            {* end(transition) *}
            {* begin(onExit) *}
            {* end(onExit) *}
            {* end(State) *}

        Stamp_states_t#StampSliderForward:
            {* begin(State) *}
            {* begin(onEntry) *}
            _transit := FALSE;
            {* end(onEntry) *}
            {* begin(onActive) *}
            StampPusher := FALSE;
            StampSliderMovedOut := TRUE;
            IF ((StampLowered = FALSE) AND (StampUp = TRUE)) THEN
                interconnect := FALSE;
            END_IF;
            Timer(IN := FALSE, PT := TIME#1.0ms);
            {* end(onActive) *}
            {* begin(transition) *}
            IF StampSliderMovedOut THEN
                _transit := TRUE;
                _state := Stamp_states_t#Step2;
            END_IF;
            {* end(transition) *}
            {* begin(onExit) *}
            {* end(onExit) *}
            {* end(State) *}

        Stamp_states_t#Stamp_Init_1:
            {* begin(State) *}
            {* begin(onEntry) *}
            _transit := FALSE;
            {* end(onEntry) *}
            {* begin(onActive) *}
            StampSliderMovedIn := TRUE;
            StampSliderMovedOut := FALSE;
            {* end(onActive) *}
            {* begin(transition) *}
            IF StampSliderSensorMovedIn THEN
                _transit := TRUE;
                _state := Stamp_states_t#Stamp_Init_2;
            END_IF;
            {* end(transition) *}
            {* begin(onExit) *}
            {* end(onExit) *}
            {* end(State) *}

        Stamp_states_t#Stamp_Init_2:
            {* begin(State) *}
            {* begin(onEntry) *}
            _transit := FALSE;
            {* end(onEntry) *}
            {* begin(onActive) *}
            StampSliderMovedIn := FALSE;
            StampSliderMovedOut := TRUE;
            {* end(onActive) *}
            {* begin(transition) *}
            IF StampSliderSensorMovedOut THEN
                _transit := TRUE;
                _state := Stamp_states_t#Stamp_Init_3;
            END_IF;
            {* end(transition) *}
            {* begin(onExit) *}
            {* end(onExit) *}
            {* end(State) *}

        Stamp_states_t#Stamp_Init_3:
            {* begin(State) *}
            {* begin(onEntry) *}
            _transit := FALSE;
            {* end(onEntry) *}
            {* begin(onActive) *}
            StampPusher := TRUE;
            {* end(onActive) *}
            {* begin(transition) *}
            IF StampLowered THEN
                _transit := TRUE;
                _state := Stamp_states_t#Stamp_Init_4;
            END_IF;
            {* end(transition) *}
            {* begin(onExit) *}
            {* end(onExit) *}
            {* end(State) *}

        Stamp_states_t#Stamp_Init_4:
            {* begin(State) *}
            {* begin(onEntry) *}
            _transit := FALSE;
            {* end(onEntry) *}
            {* begin(onActive) *}
            StampPusher := FALSE;
            {* end(onActive) *}
            {* begin(transition) *}
            IF StampUp THEN
                _transit := TRUE;
                _state := Stamp_states_t#Interstep;
            END_IF;
            {* end(transition) *}
            {* begin(onExit) *}
            {* end(onExit) *}
            {* end(State) *}

        Stamp_states_t#Start_Stamp:
            {* begin(State) *}
            {* begin(onEntry) *}
            _transit := FALSE;
            {* end(onEntry) *}
            {* begin(onActive) *}
            StampSliderMovedOut := FALSE;
            StampSliderMovedIn := FALSE;
            StampPusher := FALSE;
            StampGreenLamp := FALSE;
            StampPressure := FALSE;
            StartCommandStamp := FALSE;
            IF (StampStartButton = TRUE) THEN
                interconnectStampStartCommand := TRUE;
            END_IF;
            {* end(onActive) *}
            {* begin(transition) *}
            IF interconnectStampStartCommand THEN
                _transit := TRUE;
                _state := Stamp_states_t#Green_Lamp;
            END_IF;
            {* end(transition) *}
            {* begin(onExit) *}
            {* end(onExit) *}
            {* end(State) *}

        Stamp_states_t#Step0:
            {* begin(State) *}
            {* begin(onEntry) *}
            _transit := FALSE;
            {* end(onEntry) *}
            {* begin(onActive) *}
            {* end(onActive) *}
            {* begin(transition) *}
            IF CraneUp THEN
                _transit := TRUE;
                _state := Stamp_states_t#StampSliderBack;
            END_IF;
            {* end(transition) *}
            {* begin(onExit) *}
            {* end(onExit) *}
            {* end(State) *}

        Stamp_states_t#Step1:
            {* begin(State) *}
            {* begin(onEntry) *}
            _transit := FALSE;
            {* end(onEntry) *}
            {* begin(onActive) *}
            Timer(IN := StampLowered, PT := TIME#);
            interconnect := Timer.Q;
            {* end(onActive) *}
            {* begin(transition) *}
            IF interconnect THEN
                _transit := TRUE;
                _state := Stamp_states_t#StampSliderForward;
            END_IF;
            {* end(transition) *}
            {* begin(onExit) *}
            {* end(onExit) *}
            {* end(State) *}

        Stamp_states_t#Step2:
            {* begin(State) *}
            {* begin(onEntry) *}
            _transit := FALSE;
            {* end(onEntry) *}
            {* begin(onActive) *}
            {* end(onActive) *}
            {* begin(transition) *}
            IF (((AnalogCranePosition > INT#16160) AND (AnalogCranePosition < INT#16260)) AND NOT StampSliderFilled) THEN
                _transit := TRUE;
                _state := Stamp_states_t#Interstep;
            END_IF;
            {* end(transition) *}
            {* begin(onExit) *}
            {* end(onExit) *}
            {* end(State) *}

            END_CASE;
END_FUNCTION_BLOCK

(* ---- Scenario1v0_Final.xml.st ---- *)
TYPE
    Magazin_states_t : (Green_Lamp , Init , Interstep , Magazin_Init , Magazin_Init_2 , Slider_Move_Back , Start_Magazin , Step0 , Step1 , convey);
    Crane_states_t : (Crane_Init , Crane_Init_2 , Crane_Lift_Conveyor , Crane_Lift_Magazine , Crane_On_Conveyor , Crane_Stop , Crane_Turn_Left , Init , Interstep , Interstep_2 , Interstep_Check_Workpiece , Magazin_Stop , Start_Crane , TimeDelay , Turn_Right , release);
END_TYPE

FUNCTION_BLOCK Magazin
    VAR_INPUT  CraneDown : BOOL; END_VAR {*Irwxp*}
    VAR_INPUT  CraneOnConveyor : BOOL; END_VAR {*Irwxp*}
    VAR_INPUT  CraneOnMagazin : BOOL; END_VAR {*Irwxp*}
    VAR_INPUT  CraneSucked : BOOL; END_VAR {*Irwxp*}
    VAR_INPUT  CraneUp : BOOL; END_VAR {*Irwxp*}
    VAR_OUTPUT  MagazinGreenLamp : BOOL; END_VAR {*Orwxp*}
    VAR_OUTPUT  MagazinSlider : BOOL; END_VAR {*Orwxp*}
    VAR  SFCInit : BOOL; END_VAR {*Lrwxp*}
    VAR_INPUT  SFCReset : BOOL; END_VAR {*Irwxp*}
    VAR_INPUT  SliderMovedOut : BOOL; END_VAR {*Irwxp*}
    VAR_INPUT  SliderNotMovedOut : BOOL; END_VAR {*Irwxp*}
    VAR_INPUT  StartButtonMagazin : BOOL; END_VAR {*Irwxp*}
    VAR_OUTPUT  StartCommandMagazin : BOOL; END_VAR {*Orwxp*}
    VAR_INPUT  StartVar : BOOL; END_VAR {*Irwxp*}
    VAR_INPUT  WorkpieceReady : BOOL; END_VAR {*Irwxp*}
    VAR  _state : Magazin_states_t; END_VAR {*Lrwxp*}
    VAR  _transit : BOOL; END_VAR {*Lrwxp*}
    VAR  interconnectMagazinStartCommand : BOOL; END_VAR {*Lrwxp*}

    CASE _state OF
        Magazin_states_t#Green_Lamp:
            _transit := FALSE;
            MagazinGreenLamp := TRUE;
            interconnectMagazinStartCommand := FALSE;
            IF TRUE THEN
                _transit := TRUE;
                _state := Magazin_states_t#Magazin_Init;
            END_IF;

        Magazin_states_t#Init:
            _transit := FALSE;
            IF TRUE THEN
                _transit := TRUE;
                _state := Magazin_states_t#Start_Magazin;
            END_IF;

        Magazin_states_t#Interstep:
            _transit := FALSE;
            StartCommandMagazin := TRUE;
            IF StartVar THEN
                _transit := TRUE;
                _state := Magazin_states_t#convey;
            END_IF;

        Magazin_states_t#Magazin_Init:
            _transit := FALSE;
            MagazinSlider := TRUE;
            IF TRUE THEN
                _transit := TRUE;
                _state := Magazin_states_t#Magazin_Init_2;
            END_IF;

        Magazin_states_t#Magazin_Init_2:
            _transit := FALSE;
            MagazinSlider := FALSE;
            IF TRUE THEN
                _transit := TRUE;
                _state := Magazin_states_t#Interstep;
            END_IF;

        Magazin_states_t#Slider_Move_Back:
            _transit := FALSE;
            IF ((SliderMovedOut = TRUE) AND (SliderNotMovedOut = FALSE)) THEN
                MagazinSlider := FALSE;
            END_IF;
            IF CraneUp THEN
                _transit := TRUE;
                _state := Magazin_states_t#Step1;
            END_IF;

        Magazin_states_t#Start_Magazin:
            _transit := FALSE;
            MagazinSlider := FALSE;
            MagazinGreenLamp := FALSE;
            StartVar := FALSE;
            StartCommandMagazin := FALSE;
            IF (StartButtonMagazin = TRUE) THEN
                interconnectMagazinStartCommand := TRUE;
            END_IF;
            IF interconnectMagazinStartCommand THEN
                _transit := TRUE;
                _state := Magazin_states_t#Green_Lamp;
            END_IF;

        Magazin_states_t#Step0:
            _transit := FALSE;
            IF CraneDown THEN
                _transit := TRUE;
                _state := Magazin_states_t#Slider_Move_Back;
            END_IF;

        Magazin_states_t#Step1:
            _transit := FALSE;
            IF CraneOnConveyor THEN
                _transit := TRUE;
                _state := Magazin_states_t#Interstep;
            END_IF;

        Magazin_states_t#convey:
            _transit := FALSE;
            IF SliderNotMovedOut THEN
                MagazinSlider := TRUE;
            END_IF;
            IF CraneOnMagazin THEN
                _transit := TRUE;
                _state := Magazin_states_t#Step0;
            END_IF;

            END_CASE;
END_FUNCTION_BLOCK

PROGRAM Main

VAR  Actuator_CraneLower : BOOL; END_VAR {*Lrwxp*}
VAR  Actuator_CraneTurnClockwise : BOOL; END_VAR {*Lrwxp*}
VAR  Actuator_CraneTurnCounterclockwise : BOOL; END_VAR {*Lrwxp*}
VAR  Actuator_MagazinGreenLamp : BOOL; END_VAR {*Lrwxp*}
VAR  Actuator_MagazinSlider : BOOL; END_VAR {*Lrwxp*}
VAR  Actuator_MagazinVacuumOff : BOOL; END_VAR {*Lrwxp*}
VAR  Actuator_MagazinVacuumOn : BOOL; END_VAR {*Lrwxp*}
VAR  Actuator_MagazinWhiteLamp : BOOL; END_VAR {*Lrwxp*}
VAR  Crane : Crane; END_VAR {*Lrwxp*}
VAR  Mag : Magazin; END_VAR {*Lrwxp*}
VAR  Sensor_CraneDown : BOOL; END_VAR {*Lrwxp*}
VAR  Sensor_CraneOnConveyor : BOOL; END_VAR {*Lrwxp*}
VAR  Sensor_CraneOnMagazin : BOOL; END_VAR {*Lrwxp*}
VAR  Sensor_CranePosition : BOOL; END_VAR {*Lrwxp*}
VAR  Sensor_CraneSucked : BOOL; END_VAR {*Lrwxp*}
VAR  Sensor_CraneUp : BOOL; END_VAR {*Lrwxp*}
VAR  Sensor_MagazinEmergencyStop : BOOL; END_VAR {*Lrwxp*}
VAR  Sensor_MagazinSwitchManuellAutomatic : BOOL; END_VAR {*Lrwxp*}
VAR  Sensor_SliderMovedOut : BOOL; END_VAR {*Lrwxp*}
VAR  Sensor_SliderNotMovedOut : BOOL; END_VAR {*Lrwxp*}
VAR  Sensor_StartButtonMagazin : BOOL; END_VAR {*Lrwxp*}
VAR  Sensor_WorkpieceReady : BOOL; END_VAR {*Lrwxp*}
Mag.SliderNotMovedOut := Sensor_SliderNotMovedOut;
Mag.SliderMovedOut := Sensor_SliderMovedOut;
Mag.CraneOnMagazin := Sensor_CraneOnMagazin;
Mag.CraneDown := Sensor_CraneDown;
Mag.CraneUp := Sensor_CraneUp;
Mag.CraneOnConveyor := Sensor_CraneOnConveyor;
Mag.WorkpieceReady := Sensor_WorkpieceReady;
Mag.StartButtonMagazin := Sensor_StartButtonMagazin;
Actuator_MagazinSlider := Mag.MagazinSlider;
Actuator_MagazinGreenLamp := Mag.MagazinGreenLamp;
Crane.WorkpieceReady := Sensor_WorkpieceReady;
Crane.CraneUp := Sensor_CraneUp;
Crane.CraneOnConveyor := Sensor_CraneOnConveyor;
Crane.CraneDown := Sensor_CraneDown;
Crane.CraneSucked := Sensor_CraneSucked;
Crane.CraneOnMagazin := Sensor_CraneOnMagazin;
Crane.SliderMovedOut := Sensor_SliderMovedOut;
Crane.StartButtonMagazin := Sensor_StartButtonMagazin;
Actuator_CraneTurnCounterclockwise := Crane.CraneTurnCounterclockwise;
Actuator_CraneTurnClockwise := Crane.CraneTurnClockwise;
Actuator_CraneLower := Crane.CraneLower;
Actuator_MagazinVacuumOff := Crane.MagazinVacuumOff;
Actuator_MagazinVacuumOn := Crane.MagazinVacuumOn;
IF Sensor_MagazinEmergencyStop THEN
    Mag();
    Crane();
    IF Actuator_MagazinGreenLamp THEN
        IF (Crane.StartCommandCrane AND Mag.StartCommandMagazin) THEN
            Crane.StartVar := TRUE;
            Mag.StartVar := TRUE;
        END_IF;
    END_IF;
    Crane.SFCReset := FALSE;
    Mag.SFCReset := FALSE;
ELSEIF NOT Sensor_MagazinEmergencyStop THEN
    Actuator_MagazinSlider := FALSE;
    Actuator_CraneLower := FALSE;
    Actuator_MagazinVacuumOn := FALSE;
    Actuator_MagazinVacuumOff := TRUE;
    Actuator_MagazinGreenLamp := FALSE;
    Actuator_CraneTurnCounterclockwise := FALSE;
    Actuator_CraneTurnClockwise := FALSE;
    Crane.SFCReset := TRUE;
    Mag.SFCReset := TRUE;
    Crane.StartVar := FALSE;
    Mag.StartVar := FALSE;
END_IF;
END_PROGRAM
FUNCTION_BLOCK Crane
VAR_INPUT  CraneDown : BOOL; END_VAR {*Irwxp*}
VAR_OUTPUT  CraneLower : BOOL; END_VAR {*Orwxp*}
VAR_INPUT  CraneOnConveyor : BOOL; END_VAR {*Irwxp*}
VAR_INPUT  CraneOnMagazin : BOOL; END_VAR {*Irwxp*}
VAR_INPUT  CraneSucked : BOOL; END_VAR {*Irwxp*}
VAR_OUTPUT  CraneTurnClockwise : BOOL; END_VAR {*Orwxp*}
VAR_OUTPUT  CraneTurnCounterclockwise : BOOL; END_VAR {*Orwxp*}
VAR_INPUT  CraneUp : BOOL; END_VAR {*Irwxp*}
VAR_OUTPUT  MagazinVacuumOff : BOOL; END_VAR {*Orwxp*}
VAR_OUTPUT  MagazinVacuumOn : BOOL; END_VAR {*Orwxp*}
VAR  SFCInit : BOOL; END_VAR {*Lrwxp*}
VAR_INPUT  SFCReset : BOOL; END_VAR {*Irwxp*}
VAR_INPUT  SliderMovedOut : BOOL; END_VAR {*Irwxp*}
VAR_INPUT  SliderNotMovedOut : BOOL; END_VAR {*Irwxp*}
VAR_INPUT  StartButtonMagazin : BOOL; END_VAR {*Irwxp*}
VAR_OUTPUT  StartCommandCrane : BOOL; END_VAR {*Orwxp*}
VAR_INPUT  StartVar : BOOL; END_VAR {*Irwxp*}
VAR  TimeDelay_Timer : TON; END_VAR {*Lrwxp*}
VAR  TimeDelay_Timer_Duration : TIME := TIME#50.0ms; END_VAR {*Lrwxp*}
VAR  TimeDelay_Timer_interconnect : BOOL; END_VAR {*Lrwxp*}
VAR_INPUT  WorkpieceReady : BOOL; END_VAR {*Irwxp*}
VAR  _state : Crane_states_t; END_VAR {*Lrwxp*}
VAR  _transit : BOOL; END_VAR {*Lrwxp*}
VAR  interconnectCraneStartCommand : BOOL; END_VAR {*Lrwxp*}

CASE _state OF
    Crane_states_t#Crane_Init:
        _transit := FALSE;
        CraneLower := TRUE;
        interconnectCraneStartCommand := FALSE;
        IF CraneDown THEN
            _transit := TRUE;
            _state := Crane_states_t#Crane_Init_2;
        END_IF;

    Crane_states_t#Crane_Init_2:
        _transit := FALSE;
        CraneLower := FALSE;
        IF CraneUp THEN
            _transit := TRUE;
            _state := Crane_states_t#Interstep;
        END_IF;

    Crane_states_t#Crane_Lift_Conveyor:
        _transit := FALSE;
        CraneLower := FALSE;
        IF TRUE THEN
            _transit := TRUE;
            _state := Crane_states_t#Interstep;
        END_IF;

    Crane_states_t#Crane_Lift_Magazine:
        _transit := FALSE;
        CraneLower := FALSE;
        IF CraneUp THEN
            _transit := TRUE;
            _state := Crane_states_t#Crane_Turn_Left;
        END_IF;

    Crane_states_t#Crane_On_Conveyor:
        _transit := FALSE;
        CraneTurnCounterclockwise := FALSE;
        CraneTurnClockwise := FALSE;
        CraneLower := TRUE;
        IF CraneDown THEN
            _transit := TRUE;
            _state := Crane_states_t#release;
        END_IF;

    Crane_states_t#Crane_Stop:
        _transit := FALSE;
        IF TRUE THEN
            _transit := TRUE;
            _state := Crane_states_t#Start_Crane;
        END_IF;

    Crane_states_t#Crane_Turn_Left:
        _transit := FALSE;
        CraneTurnCounterclockwise := TRUE;
        CraneTurnClockwise := FALSE;
        IF CraneOnConveyor THEN
            _transit := TRUE;
            _state := Crane_states_t#Crane_On_Conveyor;
        END_IF;

    Crane_states_t#Init:
        _transit := FALSE;
        IF TRUE THEN
            _transit := TRUE;
            _state := Crane_states_t#Start_Crane;
        END_IF;

    Crane_states_t#Interstep:
        _transit := FALSE;
        StartCommandCrane := TRUE;
        IF StartVar THEN
            _transit := TRUE;
            _state := Crane_states_t#Interstep_2;
        END_IF;

    Crane_states_t#Interstep_2:
        _transit := FALSE;
        IF SliderMovedOut THEN
            _transit := TRUE;
            _state := Crane_states_t#TimeDelay;
        END_IF;

    Crane_states_t#Interstep_Check_Workpiece:
        _transit := FALSE;
        IF WorkpieceReady THEN
            _transit := TRUE;
            _state := Crane_states_t#Magazin_Stop;
        ELSEIF NOT WorkpieceReady THEN
            _transit := TRUE;
            _state := Crane_states_t#Crane_Stop;
        END_IF;

    Crane_states_t#Magazin_Stop:
        _transit := FALSE;
        CraneTurnClockwise := FALSE;
        CraneTurnCounterclockwise := FALSE;
        MagazinVacuumOn := TRUE;
        MagazinVacuumOff := FALSE;
        CraneLower := TRUE;
        IF CraneSucked THEN
            _transit := TRUE;
            _state := Crane_states_t#Crane_Lift_Magazine;
        END_IF;

    Crane_states_t#Start_Crane:
        _transit := FALSE;
        CraneLower := FALSE;
        MagazinVacuumOff := TRUE;
        MagazinVacuumOn := FALSE;
        CraneTurnCounterclockwise := FALSE;
        CraneTurnClockwise := FALSE;
        StartVar := FALSE;
        StartCommandCrane := FALSE;
        IF (StartButtonMagazin = TRUE) THEN
            interconnectCraneStartCommand := TRUE;
        END_IF;
        IF interconnectCraneStartCommand THEN
            _transit := TRUE;
            _state := Crane_states_t#Crane_Init;
        END_IF;

    Crane_states_t#TimeDelay:
        _transit := FALSE;
        TimeDelay_Timer(IN := TRUE, PT := TimeDelay_Timer_Duration);
        TimeDelay_Timer_interconnect := TimeDelay_Timer.Q;
        IF TimeDelay_Timer_interconnect THEN
            _transit := TRUE;
            _state := Crane_states_t#Turn_Right;
        END_IF;

    Crane_states_t#Turn_Right:
        _transit := FALSE;
        CraneTurnClockwise := TRUE;
        CraneTurnCounterclockwise := FALSE;
        IF CraneOnMagazin THEN
            _transit := TRUE;
            _state := Crane_states_t#Interstep_Check_Workpiece;
        END_IF;

    Crane_states_t#release:
        _transit := FALSE;
        MagazinVacuumOff := TRUE;
        MagazinVacuumOn := FALSE;
        IF TRUE THEN
            _transit := TRUE;
            _state := Crane_states_t#Crane_Lift_Conveyor;
        END_IF;

    END_CASE;
END_FUNCTION_BLOCK

(* ---- Scenario1v0_Final.xml_Crane.st ---- *)
FUNCTION_BLOCK Crane
    VAR_INPUT  CraneDown : BOOL; END_VAR {*Irwxp*}
    VAR_OUTPUT  CraneLower : BOOL; END_VAR {*Orwxp*}
    VAR_INPUT  CraneOnConveyor : BOOL; END_VAR {*Irwxp*}
    VAR_INPUT  CraneOnMagazin : BOOL; END_VAR {*Irwxp*}
    VAR_INPUT  CraneSucked : BOOL; END_VAR {*Irwxp*}
    VAR_OUTPUT  CraneTurnClockwise : BOOL; END_VAR {*Orwxp*}
    VAR_OUTPUT  CraneTurnCounterclockwise : BOOL; END_VAR {*Orwxp*}
    VAR_INPUT  CraneUp : BOOL; END_VAR {*Irwxp*}
    VAR_OUTPUT  MagazinVacuumOff : BOOL; END_VAR {*Orwxp*}
    VAR_OUTPUT  MagazinVacuumOn : BOOL; END_VAR {*Orwxp*}
    VAR  SFCInit : BOOL; END_VAR {*Lrwxp*}
    VAR_INPUT  SFCReset : BOOL; END_VAR {*Irwxp*}
    VAR_INPUT  SliderMovedOut : BOOL; END_VAR {*Irwxp*}
    VAR_INPUT  SliderNotMovedOut : BOOL; END_VAR {*Irwxp*}
    VAR_INPUT  StartButtonMagazin : BOOL; END_VAR {*Irwxp*}
    VAR_OUTPUT  StartCommandCrane : BOOL; END_VAR {*Orwxp*}
    VAR_INPUT  StartVar : BOOL; END_VAR {*Irwxp*}
    VAR  TimeDelay_Timer : TON; END_VAR {*Lrwxp*}
    VAR  TimeDelay_Timer_Duration : TIME := TIME#50.0ms; END_VAR {*Lrwxp*}
    VAR  TimeDelay_Timer_interconnect : BOOL; END_VAR {*Lrwxp*}
    VAR_INPUT  WorkpieceReady : BOOL; END_VAR {*Irwxp*}
    VAR  _state : Crane_states_t; END_VAR {*Lrwxp*}
    VAR  _transit : BOOL; END_VAR {*Lrwxp*}
    VAR  interconnectCraneStartCommand : BOOL; END_VAR {*Lrwxp*}

    CASE _state OF
        Crane_states_t#Crane_Init:
            _transit := FALSE;
            CraneLower := TRUE;
            interconnectCraneStartCommand := FALSE;
            IF CraneDown THEN
                _transit := TRUE;
                _state := Crane_states_t#Crane_Init_2;
            END_IF;

        Crane_states_t#Crane_Init_2:
            _transit := FALSE;
            CraneLower := FALSE;
            IF CraneUp THEN
                _transit := TRUE;
                _state := Crane_states_t#Interstep;
            END_IF;

        Crane_states_t#Crane_Lift_Conveyor:
            _transit := FALSE;
            CraneLower := FALSE;
            IF TRUE THEN
                _transit := TRUE;
                _state := Crane_states_t#Interstep;
            END_IF;

        Crane_states_t#Crane_Lift_Magazine:
            _transit := FALSE;
            CraneLower := FALSE;
            IF CraneUp THEN
                _transit := TRUE;
                _state := Crane_states_t#Crane_Turn_Left;
            END_IF;

        Crane_states_t#Crane_On_Conveyor:
            _transit := FALSE;
            CraneTurnCounterclockwise := FALSE;
            CraneTurnClockwise := FALSE;
            CraneLower := TRUE;
            IF CraneDown THEN
                _transit := TRUE;
                _state := Crane_states_t#release;
            END_IF;

        Crane_states_t#Crane_Stop:
            _transit := FALSE;
            IF TRUE THEN
                _transit := TRUE;
                _state := Crane_states_t#Start_Crane;
            END_IF;

        Crane_states_t#Crane_Turn_Left:
            _transit := FALSE;
            CraneTurnCounterclockwise := TRUE;
            CraneTurnClockwise := FALSE;
            IF CraneOnConveyor THEN
                _transit := TRUE;
                _state := Crane_states_t#Crane_On_Conveyor;
            END_IF;

        Crane_states_t#Init:
            _transit := FALSE;
            IF TRUE THEN
                _transit := TRUE;
                _state := Crane_states_t#Start_Crane;
            END_IF;

        Crane_states_t#Interstep:
            _transit := FALSE;
            StartCommandCrane := TRUE;
            IF StartVar THEN
                _transit := TRUE;
                _state := Crane_states_t#Interstep_2;
            END_IF;

        Crane_states_t#Interstep_2:
            _transit := FALSE;
            IF SliderMovedOut THEN
                _transit := TRUE;
                _state := Crane_states_t#TimeDelay;
            END_IF;

        Crane_states_t#Interstep_Check_Workpiece:
            _transit := FALSE;
            IF WorkpieceReady THEN
                _transit := TRUE;
                _state := Crane_states_t#Magazin_Stop;
            ELSEIF NOT WorkpieceReady THEN
                _transit := TRUE;
                _state := Crane_states_t#Crane_Stop;
            END_IF;

        Crane_states_t#Magazin_Stop:
            _transit := FALSE;
            CraneTurnClockwise := FALSE;
            CraneTurnCounterclockwise := FALSE;
            MagazinVacuumOn := TRUE;
            MagazinVacuumOff := FALSE;
            CraneLower := TRUE;
            IF CraneSucked THEN
                _transit := TRUE;
                _state := Crane_states_t#Crane_Lift_Magazine;
            END_IF;

        Crane_states_t#Start_Crane:
            _transit := FALSE;
            CraneLower := FALSE;
            MagazinVacuumOff := TRUE;
            MagazinVacuumOn := FALSE;
            CraneTurnCounterclockwise := FALSE;
            CraneTurnClockwise := FALSE;
            StartVar := FALSE;
            StartCommandCrane := FALSE;
            IF (StartButtonMagazin = TRUE) THEN
                interconnectCraneStartCommand := TRUE;
            END_IF;
            IF interconnectCraneStartCommand THEN
                _transit := TRUE;
                _state := Crane_states_t#Crane_Init;
            END_IF;

        Crane_states_t#TimeDelay:
            _transit := FALSE;
            TimeDelay_Timer(IN := TRUE, PT := TimeDelay_Timer_Duration);
            TimeDelay_Timer_interconnect := TimeDelay_Timer.Q;
            IF TimeDelay_Timer_interconnect THEN
                _transit := TRUE;
                _state := Crane_states_t#Turn_Right;
            END_IF;

        Crane_states_t#Turn_Right:
            _transit := FALSE;
            CraneTurnClockwise := TRUE;
            CraneTurnCounterclockwise := FALSE;
            IF CraneOnMagazin THEN
                _transit := TRUE;
                _state := Crane_states_t#Interstep_Check_Workpiece;
            END_IF;

        Crane_states_t#release:
            _transit := FALSE;
            MagazinVacuumOff := TRUE;
            MagazinVacuumOn := FALSE;
            IF TRUE THEN
                _transit := TRUE;
                _state := Crane_states_t#Crane_Lift_Conveyor;
            END_IF;

            END_CASE;
END_FUNCTION_BLOCK

(* ---- Scenario1v0_Final.xml_Magazin.st ---- *)
FUNCTION_BLOCK Magazin
    VAR_INPUT  CraneDown : BOOL; END_VAR {*Irwxp*}
    VAR_INPUT  CraneOnConveyor : BOOL; END_VAR {*Irwxp*}
    VAR_INPUT  CraneOnMagazin : BOOL; END_VAR {*Irwxp*}
    VAR_INPUT  CraneSucked : BOOL; END_VAR {*Irwxp*}
    VAR_INPUT  CraneUp : BOOL; END_VAR {*Irwxp*}
    VAR_OUTPUT  MagazinGreenLamp : BOOL; END_VAR {*Orwxp*}
    VAR_OUTPUT  MagazinSlider : BOOL; END_VAR {*Orwxp*}
    VAR  SFCInit : BOOL; END_VAR {*Lrwxp*}
    VAR_INPUT  SFCReset : BOOL; END_VAR {*Irwxp*}
    VAR_INPUT  SliderMovedOut : BOOL; END_VAR {*Irwxp*}
    VAR_INPUT  SliderNotMovedOut : BOOL; END_VAR {*Irwxp*}
    VAR_INPUT  StartButtonMagazin : BOOL; END_VAR {*Irwxp*}
    VAR_OUTPUT  StartCommandMagazin : BOOL; END_VAR {*Orwxp*}
    VAR_INPUT  StartVar : BOOL; END_VAR {*Irwxp*}
    VAR_INPUT  WorkpieceReady : BOOL; END_VAR {*Irwxp*}
    VAR  _state : Magazin_states_t; END_VAR {*Lrwxp*}
    VAR  _transit : BOOL; END_VAR {*Lrwxp*}
    VAR  interconnectMagazinStartCommand : BOOL; END_VAR {*Lrwxp*}

    CASE _state OF
        Magazin_states_t#Green_Lamp:
            _transit := FALSE;
            MagazinGreenLamp := TRUE;
            interconnectMagazinStartCommand := FALSE;
            IF TRUE THEN
                _transit := TRUE;
                _state := Magazin_states_t#Magazin_Init;
            END_IF;

        Magazin_states_t#Init:
            _transit := FALSE;
            IF TRUE THEN
                _transit := TRUE;
                _state := Magazin_states_t#Start_Magazin;
            END_IF;

        Magazin_states_t#Interstep:
            _transit := FALSE;
            StartCommandMagazin := TRUE;
            IF StartVar THEN
                _transit := TRUE;
                _state := Magazin_states_t#convey;
            END_IF;

        Magazin_states_t#Magazin_Init:
            _transit := FALSE;
            MagazinSlider := TRUE;
            IF TRUE THEN
                _transit := TRUE;
                _state := Magazin_states_t#Magazin_Init_2;
            END_IF;

        Magazin_states_t#Magazin_Init_2:
            _transit := FALSE;
            MagazinSlider := FALSE;
            IF TRUE THEN
                _transit := TRUE;
                _state := Magazin_states_t#Interstep;
            END_IF;

        Magazin_states_t#Slider_Move_Back:
            _transit := FALSE;
            IF ((SliderMovedOut = TRUE) AND (SliderNotMovedOut = FALSE)) THEN
                MagazinSlider := FALSE;
            END_IF;
            IF CraneUp THEN
                _transit := TRUE;
                _state := Magazin_states_t#Step1;
            END_IF;

        Magazin_states_t#Start_Magazin:
            _transit := FALSE;
            MagazinSlider := FALSE;
            MagazinGreenLamp := FALSE;
            StartVar := FALSE;
            StartCommandMagazin := FALSE;
            IF (StartButtonMagazin = TRUE) THEN
                interconnectMagazinStartCommand := TRUE;
            END_IF;
            IF interconnectMagazinStartCommand THEN
                _transit := TRUE;
                _state := Magazin_states_t#Green_Lamp;
            END_IF;

        Magazin_states_t#Step0:
            _transit := FALSE;
            IF CraneDown THEN
                _transit := TRUE;
                _state := Magazin_states_t#Slider_Move_Back;
            END_IF;

        Magazin_states_t#Step1:
            _transit := FALSE;
            IF CraneOnConveyor THEN
                _transit := TRUE;
                _state := Magazin_states_t#Interstep;
            END_IF;

        Magazin_states_t#convey:
            _transit := FALSE;
            IF SliderNotMovedOut THEN
                MagazinSlider := TRUE;
            END_IF;
            IF CraneOnMagazin THEN
                _transit := TRUE;
                _state := Magazin_states_t#Step0;
            END_IF;

            END_CASE;
END_FUNCTION_BLOCK
